TYPE ST_Chamber1_ServiceParam :
STRUCT
	SpinAxisJogCW : ST_Chamber1SpinAxisJogParam;
	SpinAxisMoveAbs : ST_Chamber1SpinAxisMoveAbsParam;
	SpinAxisMoveVelCW : ST_Chamber1SpinAxisMoveVelParam;
	LiftPinAxisMoveVelCW : ST_Chamber1LiftPinAxisMoveVelParam;
	LiftPinAxisMoveVelCCW : ST_Chamber1LiftPinAxisMoveVelParam;
	LiftPinAxisMoveAbs : ST_Chamber1LiftPinAxisMoveAbsParam;
	DoorClose : ST_EmptyServiceParam;
	DoorOpen : ST_EmptyServiceParam;
	VacuumOn : ST_EmptyServiceParam;
	VacuumOff : ST_EmptyServiceParam;
	PreparePosition : ST_Chamber1PreparePositionParam;
	Endpoint1PrepareSendWafer : ST_EmptyServiceParam;
	SetMaterialParam : ST_MaterialParam;
END_STRUCT
END_TYPE

(* stored: Version 1.1.0.1, ProductVersion 3.1.4026.18
   DUT ST_Chamber1_ServiceParam: Id {9d771c70-165f-48ed-a888-a145a70861d4} *)
